// TIA Portal project "PLCSIM15-Comparison Function_V16" (V16)
// Vorlageprojekt für das Buch mit Zielsystem S7-1200

(* hardware
DEVICE "S7-1200-Station_1"  S7-1200 Station
   slot 0: "Baugruppenträger_0"  Rack  V1.0
   slot 1: "PLC_1"  CPU 1214C DC/DC/DC  6ES7 214-1AG40-0XB0  V4.0
DEVICE "HMI_1"  TP700 Comfort
   slot 0: "HMI_1"  TP700 Comfort  6AV2 124-0GC01-0AX0  16.0.0.0
   slot 1: "HMI_RT_1"  TP700 Comfort  6AV2 124-0GC01-0AX0  16.0.0.0
   slot 5: "HMI_1.IE_CP_1"  PROFINET Interface  16.0.0.0
      slot 1: "PROFINET Interface_1"  PROFINET Interface
         slot 1: "Port_1"  Port
         slot 2: "Port_2"  Port
   slot 7: "HMI_1.MPI/DP_CP_1"  MPI/DP Interface  16.0.0.0
*)

// ===== PLC "PLC_1"  CPU 1214C DC/DC/DC =====

VAR_GLOBAL   // PLC tag table "Standard-Variablentabelle"
   "FIO_LOW_LEVEL" AT %M0.0 : Bool;
   "FIO_HIGH_LEVEL" AT %M0.1 : Bool;
   "FIO_FILL_VALVE" AT %Q0.0 : Bool;
   "FIO_DISCHARGE_VALVE" AT %Q0.1 : Bool;
   "BUTTON_START" AT %I0.0 : Bool;
   "BUTTON_STOP" AT %I0.1 : Bool;
   "SWITCHER_MODE_SEL" AT %I0.4 : Bool;
   "BUTTON_MAN_FILL" AT %I1.0 : Bool;
   "BUTTON_MAN_DISCH" AT %I1.1 : Bool;
   "BUTTON_E_STOP" AT %I0.2 : Bool;
   "HMI_LAMP_RUN" AT %M12.0 : Bool;
   "HMI_LAMP_AUTO" AT %M12.1 : Bool;
   "HMI_LAMP_ESTOP" AT %M12.3 : Bool;
   "SYS_RUNNING" AT %M20.0 : Bool;
   "SEQ_PUMPING" AT %M20.1 : Bool;
   "SEQ_DRAINING" AT %M20.2 : Bool;
   "HMI_LAMP_MAN" AT %M12.2 : Bool;
   "Tag_1" AT %QW30 : Int;
   "Tag_2" AT %QW32 : Int;
   "Tag_3" AT %IW30 : Int;
   "SYS_EMERGENCY" AT %M20.3 : Bool;
   "BUTTON_RESET" AT %I0.3 : Bool;
   "CHUAN_HOA" AT %MD100 : Real;
   "MUCNUOCTHUCTE" AT %MD104 : Real;
   "MUCNUOCTHAP_HMI" AT %MD114 : Real;
   "MUCNUOCCAO_HMI" AT %MD110 : Real;
   "SYS_READY" AT %M2.0 : Bool;
END_VAR

FUNCTION "MHJ-PLC-Lab-Function-S71200" : Void   // FC9000, SCL
{ S7_Optimized_Access := 'TRUE' }
VERSION : 0.1
   VAR_TEMP
      rdTimeReturn : Int;
      outputTime : DTL;
      SyncVal : Byte;
      forVal : Int;
      forVal_2 : Int;
      Value : Byte;
   END_VAR
   VAR CONSTANT
      CompVal : Byte := 16#34;
      Value_01 : Byte := 16#11;
      Value_01_DW : DWord := 16#A165_D992;
      Value_02_DW : DWord := 16#58BE_4401;
   END_VAR
BEGIN

   #Value:=PEEK(area := 16#82,
        dbNumber := 0,
        byteOffset := 511);
   #Value := #Value + 1;

   POKE(area := 16#82,
        dbNumber := 0,
        byteOffset := 511,
        value := #Value);

   POKE(area:=16#81,
        dbNumber:=0,
        byteOffset:=1016,
        value:=#Value_01_DW);
   POKE(area := 16#81,
        dbNumber := 0,
        byteOffset := 1020,
        value := #Value_02_DW);

   POKE(area := 16#81,
        dbNumber := 0,
        byteOffset := 511,
        value := B#16#00);

   FOR #forVal := 0 TO 120 DO
       FOR #forVal_2:=0 TO 10 DO
           #rdTimeReturn:=RD_SYS_T(#outputTime);
           #rdTimeReturn := WR_SYS_T(#outputTime);
           #rdTimeReturn := RD_SYS_T(#outputTime);
           #rdTimeReturn := WR_SYS_T(#outputTime);
       END_FOR;
       #SyncVal:= PEEK(area := 16#81,
                      dbNumber := 0,
                      byteOffset := 511);
       IF #SyncVal = #CompVal THEN
          GOTO M_1;
       END_IF;
   END_FOR;
   RETURN;

   M_1:
   POKE(area := 16#81,
        dbNumber := 0,
        byteOffset := 511,
        value := B#16#0);
END_FUNCTION

ORGANIZATION_BLOCK "Main"   // OB1, LAD, ProgramCycle
TITLE = "Main Program Sweep (Cycle)"
{ S7_Optimized_Access := 'TRUE' }
VERSION : 0.1
   VAR_INPUT
      Initial_Call : Bool;   // Initial call of this OB
      Remanence : Bool;   // =True, if remanent data are available
   END_VAR
   VAR_TEMP
      Clock_1Hz : Bool;
   END_VAR
BEGIN

REGION Network 1: Connection block for PLCSIM communications. Don't delete this network! / BLOCK KẾT NỐI MÔ PHỎNG CÓ SẴN
   // Im Netzwerk 1 wird der Konnektierungsbaustein für PLC-Lab aufgerufen.
   // Dieser Aufruf darf nicht entfernt werden!
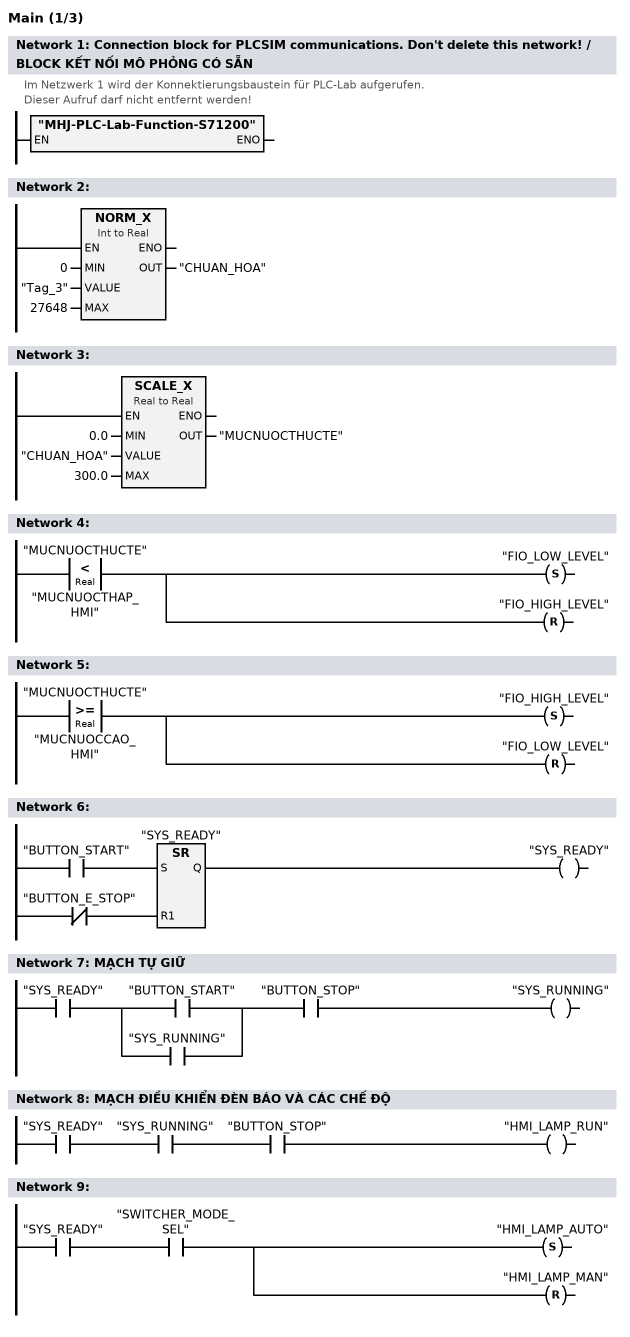
   RUNG wire#powerrail
      "MHJ-PLC-Lab-Function-S71200"()
   END_RUNG
   // the same network as SCL:
   "MHJ-PLC-Lab-Function-S71200"();
END_REGION

REGION Network 2
   RUNG wire#powerrail
      { S7_Templates := "[SrcType := Int, DestType := Real]" } Normalize(min := 0, value := "Tag_3", max := 27648, out => "CHUAN_HOA")
   END_RUNG
   // the same network as SCL:
   "CHUAN_HOA" := NORM_X(MIN := 0, VALUE := "Tag_3", MAX := 27648);
END_REGION

REGION Network 3
   RUNG wire#powerrail
      { S7_Templates := "[SrcType := Real, DestType := Real]" } Scale(min := 0.0, value := "CHUAN_HOA", max := 300.0, out => "MUCNUOCTHUCTE")
   END_RUNG
   // the same network as SCL:
   "MUCNUOCTHUCTE" := SCALE_X(MIN := 0.0, VALUE := "CHUAN_HOA", MAX := 300.0);
END_REGION

REGION Network 4
   RUNG wire#powerrail
      { S7_Templates := "SrcType := Real" } LT_Contact(in1 := "MUCNUOCTHUCTE", in2 := "MUCNUOCTHAP_HMI")
      wire#w1
      S_Coil( "FIO_LOW_LEVEL" )
   END_RUNG
   RUNG wire#w1
      R_Coil( "FIO_HIGH_LEVEL" )
   END_RUNG
   // the same network as SCL:
   IF "MUCNUOCTHUCTE" < "MUCNUOCTHAP_HMI" THEN
       "FIO_LOW_LEVEL" := TRUE;
       "FIO_HIGH_LEVEL" := FALSE;
   END_IF;
END_REGION

REGION Network 5
   RUNG wire#powerrail
      { S7_Templates := "SrcType := Real" } GE_Contact(in1 := "MUCNUOCTHUCTE", in2 := "MUCNUOCCAO_HMI")
      wire#w1
      S_Coil( "FIO_HIGH_LEVEL" )
   END_RUNG
   RUNG wire#w1
      R_Coil( "FIO_LOW_LEVEL" )
   END_RUNG
   // the same network as SCL:
   IF "MUCNUOCTHUCTE" >= "MUCNUOCCAO_HMI" THEN
       "FIO_HIGH_LEVEL" := TRUE;
       "FIO_LOW_LEVEL" := FALSE;
   END_IF;
END_REGION

REGION Network 6
   RUNG wire#powerrail
      Contact( "BUTTON_START" )
      S_SR(operand := "SYS_READY", r1 := wire#w1)
      Coil( "SYS_READY" )
   END_RUNG
   RUNG wire#powerrail
      I_Contact( "BUTTON_E_STOP" )
   END_RUNG wire#w1
   // the same network as SCL:
   IF "BUTTON_START" THEN
       "SYS_READY" := TRUE;   // SR flip-flop
   END_IF;
   IF NOT "BUTTON_E_STOP" THEN "SYS_READY" := FALSE; END_IF;
   "SYS_READY" := "SYS_READY";
END_REGION

REGION Network 7: MẠCH TỰ GIỮ
   RUNG wire#powerrail
      Contact( "SYS_READY" )
      wire#w1
      Contact( "BUTTON_START" )
      wire#w2
      Contact( "BUTTON_STOP" )
      Coil( "SYS_RUNNING" )
   END_RUNG
   RUNG wire#w1
      Contact( "SYS_RUNNING" )
   END_RUNG wire#w2
   // the same network as SCL:
   "SYS_RUNNING" := "SYS_READY" AND ("BUTTON_START" OR "SYS_RUNNING") AND "BUTTON_STOP";
END_REGION

REGION Network 8: MẠCH ĐIỀU KHIỂN ĐÈN BÁO VÀ CÁC CHẾ ĐỘ
   RUNG wire#powerrail
      Contact( "SYS_READY" )
      Contact( "SYS_RUNNING" )
      Contact( "BUTTON_STOP" )
      Coil( "HMI_LAMP_RUN" )
   END_RUNG
   // the same network as SCL:
   "HMI_LAMP_RUN" := "SYS_READY" AND "SYS_RUNNING" AND "BUTTON_STOP";
END_REGION

REGION Network 9
   RUNG wire#powerrail
      Contact( "SYS_READY" )
      Contact( "SWITCHER_MODE_SEL" )
      wire#w1
      S_Coil( "HMI_LAMP_AUTO" )
   END_RUNG
   RUNG wire#w1
      R_Coil( "HMI_LAMP_MAN" )
   END_RUNG
   // the same network as SCL:
   IF "SYS_READY" AND "SWITCHER_MODE_SEL" THEN
       "HMI_LAMP_AUTO" := TRUE;
       "HMI_LAMP_MAN" := FALSE;
   END_IF;
END_REGION

REGION Network 10
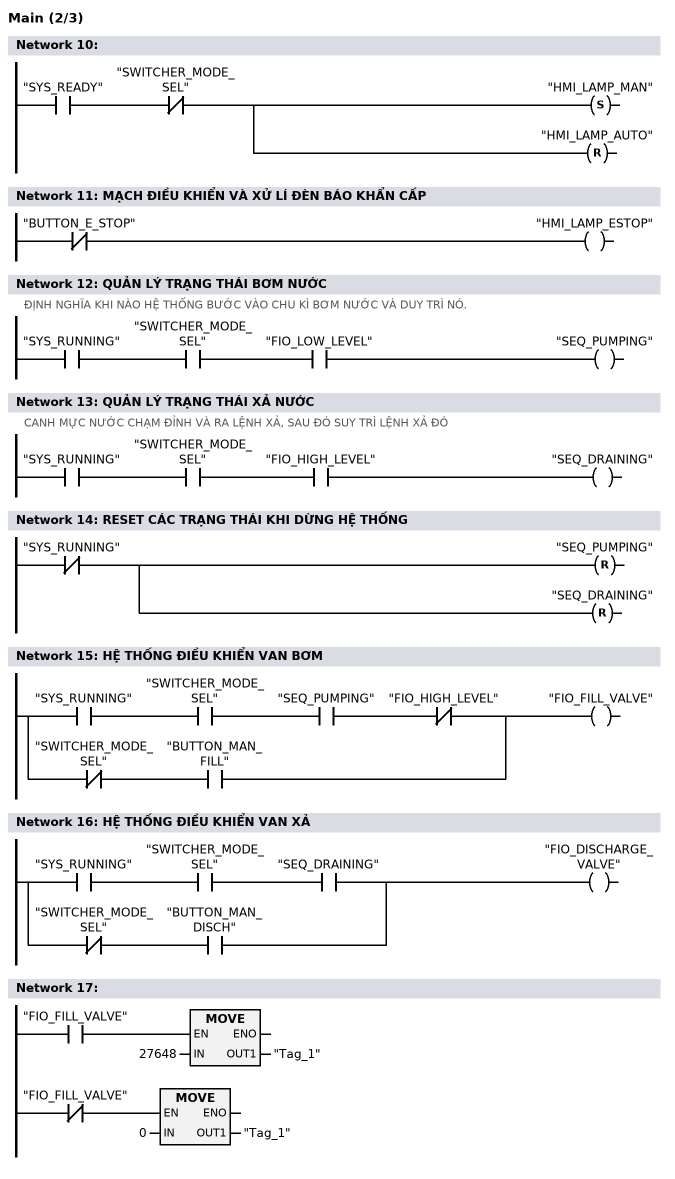
   RUNG wire#powerrail
      Contact( "SYS_READY" )
      I_Contact( "SWITCHER_MODE_SEL" )
      wire#w1
      S_Coil( "HMI_LAMP_MAN" )
   END_RUNG
   RUNG wire#w1
      R_Coil( "HMI_LAMP_AUTO" )
   END_RUNG
   // the same network as SCL:
   IF "SYS_READY" AND NOT "SWITCHER_MODE_SEL" THEN
       "HMI_LAMP_MAN" := TRUE;
       "HMI_LAMP_AUTO" := FALSE;
   END_IF;
END_REGION

REGION Network 11: MẠCH ĐIỀU KHIỂN VÀ XỬ LÍ ĐÈN BÁO KHẨN CẤP
   RUNG wire#powerrail
      I_Contact( "BUTTON_E_STOP" )
      Coil( "HMI_LAMP_ESTOP" )
   END_RUNG
   // the same network as SCL:
   "HMI_LAMP_ESTOP" := NOT "BUTTON_E_STOP";
END_REGION

REGION Network 12: QUẢN LÝ TRẠNG THÁI BƠM NƯỚC
   // ĐỊNH NGHĨA KHI NÀO HỆ THỐNG BƯỚC VÀO CHU KÌ BƠM NƯỚC VÀ DUY TRÌ NÓ.
   RUNG wire#powerrail
      Contact( "SYS_RUNNING" )
      Contact( "SWITCHER_MODE_SEL" )
      Contact( "FIO_LOW_LEVEL" )
      Coil( "SEQ_PUMPING" )
   END_RUNG
   // the same network as SCL:
   "SEQ_PUMPING" := "SYS_RUNNING" AND "SWITCHER_MODE_SEL" AND "FIO_LOW_LEVEL";
END_REGION

REGION Network 13: QUẢN LÝ TRẠNG THÁI XẢ NƯỚC
   // CANH MỰC NƯỚC CHẠM ĐỈNH VÀ RA LỆNH XẢ, SAU ĐÓ SUY TRÌ LỆNH XẢ ĐÓ
   RUNG wire#powerrail
      Contact( "SYS_RUNNING" )
      Contact( "SWITCHER_MODE_SEL" )
      Contact( "FIO_HIGH_LEVEL" )
      Coil( "SEQ_DRAINING" )
   END_RUNG
   // the same network as SCL:
   "SEQ_DRAINING" := "SYS_RUNNING" AND "SWITCHER_MODE_SEL" AND "FIO_HIGH_LEVEL";
END_REGION

REGION Network 14: RESET CÁC TRẠNG THÁI KHI DỪNG HỆ THỐNG
   RUNG wire#powerrail
      I_Contact( "SYS_RUNNING" )
      wire#w1
      R_Coil( "SEQ_PUMPING" )
   END_RUNG
   RUNG wire#w1
      R_Coil( "SEQ_DRAINING" )
   END_RUNG
   // the same network as SCL:
   IF NOT "SYS_RUNNING" THEN
       "SEQ_PUMPING" := FALSE;
       "SEQ_DRAINING" := FALSE;
   END_IF;
END_REGION

REGION Network 15: HỆ THỐNG ĐIỀU KHIỂN VAN BƠM
   RUNG wire#powerrail
      Contact( "SYS_RUNNING" )
      Contact( "SWITCHER_MODE_SEL" )
      Contact( "SEQ_PUMPING" )
      I_Contact( "FIO_HIGH_LEVEL" )
      wire#w1
      Coil( "FIO_FILL_VALVE" )
   END_RUNG
   RUNG wire#powerrail
      I_Contact( "SWITCHER_MODE_SEL" )
      Contact( "BUTTON_MAN_FILL" )
   END_RUNG wire#w1
   // the same network as SCL:
   "FIO_FILL_VALVE" := ("SYS_RUNNING" AND "SWITCHER_MODE_SEL" AND "SEQ_PUMPING" AND NOT "FIO_HIGH_LEVEL") OR (NOT "SWITCHER_MODE_SEL" AND "BUTTON_MAN_FILL");
END_REGION

REGION Network 16: HỆ THỐNG ĐIỀU KHIỂN VAN XẢ
   RUNG wire#powerrail
      Contact( "SYS_RUNNING" )
      Contact( "SWITCHER_MODE_SEL" )
      Contact( "SEQ_DRAINING" )
      wire#w1
      Coil( "FIO_DISCHARGE_VALVE" )
   END_RUNG
   RUNG wire#powerrail
      I_Contact( "SWITCHER_MODE_SEL" )
      Contact( "BUTTON_MAN_DISCH" )
   END_RUNG wire#w1
   // the same network as SCL:
   "FIO_DISCHARGE_VALVE" := ("SYS_RUNNING" AND "SWITCHER_MODE_SEL" AND "SEQ_DRAINING") OR (NOT "SWITCHER_MODE_SEL" AND "BUTTON_MAN_DISCH");
END_REGION

REGION Network 17
   RUNG wire#powerrail
      Contact( "FIO_FILL_VALVE" )
      Move(in := 27648, out1 => "Tag_1")
   END_RUNG
   RUNG wire#powerrail
      I_Contact( "FIO_FILL_VALVE" )
      Move(in := 0, out1 => "Tag_1")
   END_RUNG
   // the same network as SCL:
   IF "FIO_FILL_VALVE" THEN "Tag_1" := 27648; END_IF;
   IF NOT "FIO_FILL_VALVE" THEN "Tag_1" := 0; END_IF;
END_REGION

REGION Network 18
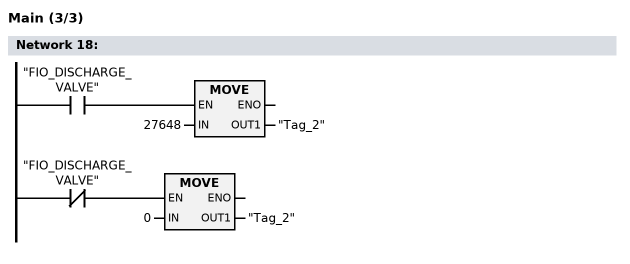
   RUNG wire#powerrail
      Contact( "FIO_DISCHARGE_VALVE" )
      Move(in := 27648, out1 => "Tag_2")
   END_RUNG
   RUNG wire#powerrail
      I_Contact( "FIO_DISCHARGE_VALVE" )
      Move(in := 0, out1 => "Tag_2")
   END_RUNG
   // the same network as SCL:
   IF "FIO_DISCHARGE_VALVE" THEN "Tag_2" := 27648; END_IF;
   IF NOT "FIO_DISCHARGE_VALVE" THEN "Tag_2" := 0; END_IF;
END_REGION
END_ORGANIZATION_BLOCK

(* ===== HMI "HMI_RT_1" =====
system functions are stored by id; their names below are inferred from use
connection "HMI_Connection_1": ETHERNET, S7_1200_OMS

HMI tags "Default tag table"
   "Tag_ScreenNumber" : UInt, internal
   "HMI_MUCNUOC" : Real = PLC MUCNUOCTHUCTE AT %MD104, 1 s
   "HMI_MUCNUOCCAOSP" : Real = PLC MUCNUOCCAO_HMI AT %MD110, 1 s
   "HMI_MUCNUOCTHAPSP" : Real = PLC MUCNUOCTHAP_HMI AT %MD114, 1 s
   "HMI_LAMP_RUN" : Bool = PLC HMI_LAMP_RUN AT %M12.0, 1 s
   "HMI_LAMP_AUTO" : Bool = PLC HMI_LAMP_AUTO AT %M12.1, 1 s
   "HMI_LAMP_ESTOP" : Bool = PLC HMI_LAMP_ESTOP AT %M12.3, 1 s
   "HMI_LAMP_MAN" : Bool = PLC HMI_LAMP_MAN AT %M12.2, 1 s

screen "Root screen" 800x420, template "Template_1"
   on GenerateScreen: SetTag("Tag_ScreenNumber", 1)
   Bar "Bar_1" at 349,68 size 172x285; MinimumValue 0; MaximumValue 300
      ProcessValue <- "HMI_MUCNUOC"
   IOField "I/O field_1" at 229,204 size 96x32; FormatPattern 999.9
      ProcessValue <- "HMI_MUCNUOC"
   IOField "I/O field_2" at 229,321 size 96x32; FormatPattern 999.9
      ProcessValue <- "HMI_MUCNUOCTHAPSP"
   IOField "I/O field_3" at 229,70 size 96x32; FormatPattern 999.9
      ProcessValue <- "HMI_MUCNUOCCAOSP"
   Circle "Circle_1" at 552,58 size 109x109
      Appearance <- "HMI_LAMP_RUN"
   TextField "Text field_1" at 71,80 size 145x22; Text 'HIGH SETPOINT'
   TextField "Text field_2" at 71,330 size 140x22; Text 'LOW SETPOINT'
   TextField "Text field_3" at 63,214 size 153x22; Text 'REAL-TIME LEVEL'
   Circle "Circle_2" at 689,58 size 108x108
      Appearance <- "HMI_LAMP_ESTOP"
   Circle "Circle_3" at 558,232 size 111x111
      Appearance <- "HMI_LAMP_AUTO"
   Circle "Circle_4" at 686,232 size 111x111
      Appearance <- "HMI_LAMP_MAN"
   TextField "Text field_4" at 586,99 size 44x23; Text 'RUN'
   TextField "Text field_5" at 712,99 size 64x23; Text 'ESTOP'
   TextField "Text field_6" at 586,275 size 56x23; Text 'AUTO'
   TextField "Text field_7" at 705,275 size 82x23; Text 'MANUAL'
   TextField "Text field_8" at 233,7 size 422x32; Text 'WATER LEVEL CONTROL SYSTEM'

Template "Template_1" 800x420
   Button "Template_Button" at 720,360 size 78x58; TextOff 'Text'
   Button "Template_Button_1" at 640,360 size 78x58; TextOff 'Text'
   Button "Template_Button_2" at 560,360 size 78x58; TextOff 'Text'
   Button "Template_Button_3" at 480,360 size 78x58; TextOff 'Text'
   Button "Template_Button_4" at 400,360 size 78x58; TextOff 'Text'
   Button "Template_Button_5" at 321,360 size 78x58; TextOff 'Text'
   Button "Template_Button_6" at 241,360 size 78x58; TextOff 'Text'
   Button "Template_Button_7" at 161,360 size 78x58; TextOff 'Text'
   Button "Template_Button_8" at 81,360 size 78x58; TextOff 'Text'
   Button "Alarms" at 1,360 size 78x58; TextOff 'Alarms'; PictureOff "AlarmDisplay_TP700_Comfort_TR"; PictureOn "AlarmDisplay_TP700_Comfort_TR"
      on Release: function_ef3f5d25("Alarm window_Unacknowledged", -1)
*)